// TwinCAT 3 PLC project Untitled1
// ProgramVersion: 3.1.4023.0
// libraries:
//   Tc2_MC2, * (Beckhoff Automation GmbH)
//   Tc2_Standard, * (Beckhoff Automation GmbH)
//   Tc2_System, * (Beckhoff Automation GmbH)
//   Tc3_Module, * (Beckhoff Automation GmbH)
// project tree:
//   / PlcTask.TcTTO
//   POUs/ MAIN.TcPOU
// real-time tasks:
//   TASK PlcTask: cycle T#10ms, priority 20, ADS port 350
// motion (NC):
//   TASK NC-Task 1 SAF: cycle T#2ms, priority 4, ADS port 501
//   TASK NC-Task 1 SVB: cycle T#10ms, priority 8, ADS port 511
//   AXIS Axis 1 (id 1)
//     OtherSettings: AllowMotionCmdToSlave=true
//     encoder EncType=1
//     drive DrvType=5
//       Analog: TorqueSetpointScale=10, ScaleFactorActTorque=0.1
//     controller CtrType=1
//       CtrPara: PriorControlFactor=1
//         Observer: BandWidth=20
// variable links:
//   Untitled1/Untitled1 Instance <-> NC-Task 1 SAF/Axes/Axis 1
//     PlcTask Inputs/MAIN.Axis.NcToPlc <-> Outputs/ToPlc
//     PlcTask Outputs/MAIN.Axis.PlcToNc <-> Inputs/FromPlc

CONFIGURATION Untitled1
    RESOURCE PLC ON TwinCAT3
        TASK PlcTask(INTERVAL := T#10ms, PRIORITY := 20);
        PROGRAM MAIN WITH PlcTask : MAIN;
    END_RESOURCE
END_CONFIGURATION

// ---- POUs/MAIN.TcPOU
PROGRAM MAIN
VAR
	Axis			:	AXIS_REF;

	fbPower			:	MC_Power;
	bEnable			:	BOOL;
	bIsAxisReady	:	BOOL;
	
	fbMoveAbsolute	:	MC_MoveAbsolute;
	bExecute		:	BOOL;
	fPosition		:	LREAL;
	fVelocity		:	LREAL;
	bBusy			:	BOOL;
	bDone			:	bool;
END_VAR

Axis(); // Axis 정보 갱신

fbPower(
	Axis := Axis,
	Enable := bEnable,
	Enable_Positive := bEnable,
	Enable_Negative := bEnable,
	Status => bIsAxisReady // Axis가 동작할 준비가 왼료되면 TRUE
);

fbMoveAbsolute(
	Axis := Axis,
	Execute := bExecute,
	Position := fPosition,
	Velocity := fVelocity,
	Busy => bBusy,
	Done => bDone 
);

END_PROGRAM
